Fanuc KAREL source: kt00145.KL

-- PROVISIONAL review KL for V770-1; original PC SHA256 3b8be3963bd63feb59ad232c4a164c2799d4abc2cd932ebd03de3cf3fb6dc5e6
-- Incomplete behavior may be omitted. Consult companion uncertainty JSON. Do not deploy.
PROGRAM KT00145
%NOLOCKGROUP
VAR
  I2 : INTEGER
  OUT : INTEGER
-- UNRESOLVED_DECL Y1 type=002018
BEGIN
  -- UNRESOLVED_PC offsets 5-19; opcodes 2E,22,9D,33,B2
  -- UNRESOLVED_PC offsets 24-35; opcodes 2E,23
  -- UNRESOLVED_PC offsets 40-62; opcodes 22,9D,33,B1,21,55,23
  -- UNRESOLVED_PC offsets 67-71; opcodes 7F
END KT00145
